{attribute 'enable_dynamic_creation'}
TYPE NodeST :
STRUCT
	data : ListItem;
	next : POINTER TO Node;
END_STRUCT
END_TYPE

(* stored: Version 1.1.0.1, ProductVersion 3.1.4024.11
   DUT NodeST: Id {0faa8581-79c5-44ce-9500-64673d67c97e} *)
